(* PLC project WAVE_TEST, Actility iec 1.0 *)
(* stored: creationDateTime 2013-01-02T13:55:36, modificationDateTime 2013-04-22T03:51:23 *)

PROGRAM main
  VAR
    AV : REAL := 100;
    AMP : REAL := 10;
    P : REAL := 30;
    SIG : INT := 1;
    V : REAL;
    Wave1 : WAVE_GENERATOR;
  END_VAR
  VAR_EXTERNAL
    GLO1 : REAL;
    GLO2 : DINT;
  END_VAR
  VAR
    REP AT %OX2.1 : BOOL;
  END_VAR
  VAR
    HYSTERESIS0 : HYSTERESIS;
    XIN2 : REAL := 10;
    EPS : REAL := 10;
  END_VAR

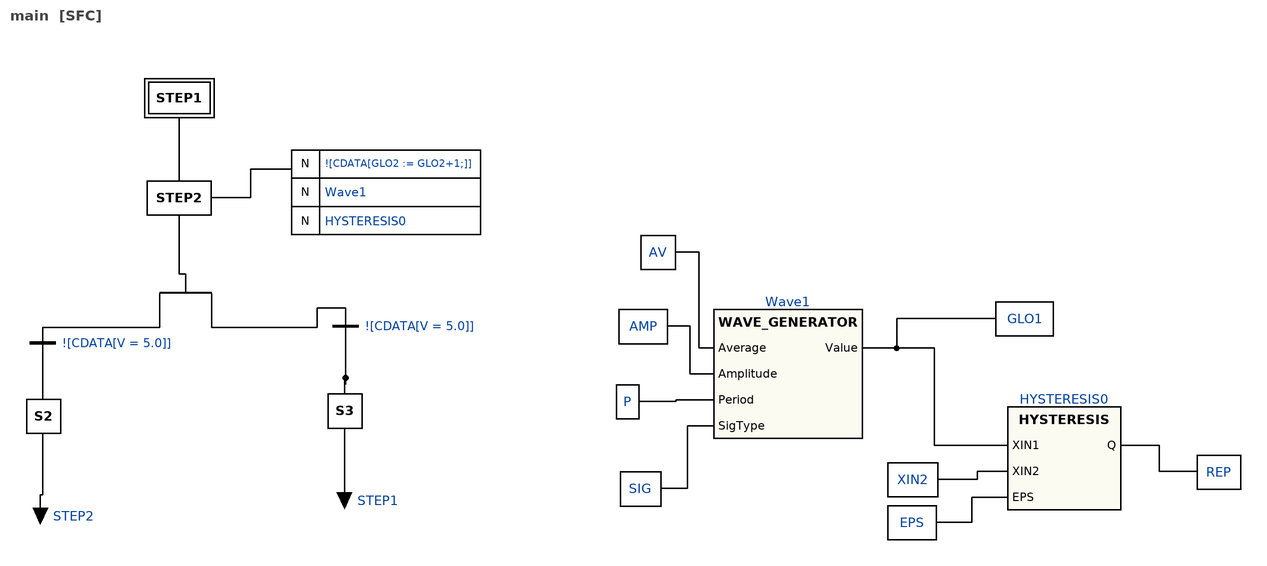
INITIAL_STEP STEP1:
  COMPUTE_FUNCTION_BLOCKS(S);
END_STEP
STEP STEP2:
  STEP2_INLINE1(N);
  Wave1(N);
  HYSTERESIS0(N);
END_STEP
ACTION STEP2_INLINE1:
  ![CDATA[GLO2 := GLO2+1;]]
END_ACTION
TRANSITION FROM STEP2 TO S2
  := ![CDATA[V = 5.0]];
END_TRANSITION
TRANSITION FROM STEP2 TO S3
  := ![CDATA[V = 5.0]];
END_TRANSITION
STEP S3:
END_STEP
STEP S2:
END_STEP
ACTION COMPUTE_FUNCTION_BLOCKS:  (* blocks drawn on the SFC sheet *)
  Wave1(Average := AV, Amplitude := AMP, Period := P, SigType := SIG);
  GLO1 := Wave1.Value;
  HYSTERESIS0(XIN1 := Wave1.Value, XIN2 := XIN2, EPS := EPS);
  REP := HYSTERESIS0.Q;
END_ACTION
END_PROGRAM

CONFIGURATION STD_CONF
  VAR_GLOBAL RETAIN
    GLO1 AT %OX1.1 : REAL := 11;
  END_VAR
  VAR_GLOBAL
    TempRoom1 AT %IX1.1 : REAL;
    TempRoom2 AT %IX1.2 : REAL;
    SumConso AT %IX0.0 : REAL;
    OnOffStatus AT %IX0.1 : REAL;
    InstantConso AT %IX0.3 : REAL;
  END_VAR
  RESOURCE STD_RESSOURCE ON PLC
    VAR_GLOBAL RETAIN
      GLO2 : DINT := 22;
    END_VAR
    TASK task2(INTERVAL := T#5s0ms, PRIORITY := 0);
    PROGRAM instance2 WITH task2 : main;
  END_RESOURCE
  RESOURCE resource0 ON PLC
  END_RESOURCE
END_CONFIGURATION
